{attribute 'qualified_only'}
VAR_GLOBAL
END_VAR

(* stored: Version 1.1.0.1, ProductVersion 3.1.4024.10
   GVL G_Sensors: Id {d28c946e-63b0-41ab-8fee-be9b6a0df66e} *)
